// TIA Portal V19 export
TYPE "PPrf_CoilHandling_MaterialFeeding"
// stored: Access Published
   STRUCT
      DecoilerFeedMode { S7_SetPoint := 'True'} : UInt;   // 0=Pneumatic braking; 1=Motor Feeding
      StraightenerRollsUse { S7_SetPoint := 'True'} : UInt;
      Vel { S7_SetPoint := 'True'} : LReal;   // [mm/min] Default value if Actual PPrg.Gen.CycleTime <= 0
      Acc { S7_SetPoint := 'True'} : LReal;   // [mm/s²] Acceleration of the material fed by straightener & decoiler
      Dec { S7_SetPoint := 'True'} : LReal;   // [mm/s²] Deceleration of the material fed by straightener & decoiler
      Jerk { S7_SetPoint := 'True'} : LReal;   // [mm/s³]
   END_STRUCT;
END_TYPE
